SUBAPPLICATION SoftKey_Kurz_Lang (* Unterscheidet kurzen Tastendruck (Loslassen vor Ablauf PT) von langem Tastendruck (PT gehalten) auf einem AX-Adapter-Eingang (z.B. Softkey_IXA.IN). LANG feuert sofort beim Erreichen von PT (nicht erst beim Loslassen); KURZ feuert beim Loslassen, wenn PT noch nicht erreicht war. PT konfigurierbar (Parameter, Default 5s). *)
  (* Standard: 61499-2; Description: Copyright (c) 2026 Meisterschulen am Ostbahnhof This program and the accompanying materials are made available under the terms of the Eclipse Public License 2.0 which is available at https://www.eclipse.org/legal/epl-2.0/ SPDX-License-Identifier: EPL-2.0 *)
  (* Version 2.0, 2026-09-11, Franz Höpfinger, Meisterschulen am Ostbahnhof, PT konfigurierbar gemacht (Parameter statt fest 5s), umbenannt von SoftKey_Kurz_Lang_5s. Race-Bug behoben: PERMIT_KURZ pruefte bisher E_TON.Q im selben Loslass-Event, das E_TON.Q durch denselben IN-Flankenwechsel bereits auf FALSE zuruecksetzt - KURZ waere dadurch IMMER durchgelassen worden, auch nach bereits gefeuertem LANG (Ausfuehrungsreihenfolge zwischen E_TON und F_TRIG_RELEASE auf denselben IN-Event ist nicht garantiert/nicht das Kriterium). Neu: eigener LANG_LATCH (AX_SR), gesetzt durch R_TRIG_LONG (waehrend PT noch gehalten wird, zeitlich klar vor jedem Loslassen), zurueckgesetzt erst beim naechsten Tastendruck-Start (R_TRIG_PRESS) - PERMIT_KURZ prueft jetzt diesen Latch statt E_TON.Q direkt. Ausserdem SPLIT_IN (AX_SPLIT_3) ergaenzt: IN wird auf 3 Sockets (E_TON/R_TRIG_PRESS/F_TRIG_RELEASE) verteilt - ein AX-Socket darf nicht direkt auf mehrere Ziel-Sockets verbunden werden, dafuer gibt es die AX_SPLIT_n-Familie. *)
  (* Version 1.0, 2026-09-11, Franz Höpfinger, Meisterschulen am Ostbahnhof, initial implementation - fuer Achslenkung-Mittelpunkt-Taste (kurz=Anfahren, lang=Speichern), generisch fuer jede Softkey-Kurz/Lang-Unterscheidung *)
  PACKAGE MyLib::sys;
  (* Documentation:
  Kurz/Lang-Druck-Unterscheidung (konfigurierbare Haltezeit)
   E_TON (AX_TON, PT als Parameter/InputVar konfigurierbar, Default 5s) laeuft solange IN gehalten wird. R_TRIG_LONG erkennt die steigende Flanke von E_TON.Q - das ist der Moment, in dem PT erreicht ist, waehrend die Taste noch gehalten wird - und feuert LANG sofort, ohne auf das Loslassen zu warten. Gleichzeitig setzt R_TRIG_LONG den LANG_LATCH (AX_SR).
   F_TRIG_RELEASE erkennt die fallende Flanke von IN (Loslassen). PERMIT_KURZ (AX_E_PERMIT_INVERT_1) laesst dieses Ereignis nur durch, wenn LANG_LATCH.Q zu diesem Zeitpunkt FALSE ist - also wenn LANG in diesem Tastendruck-Zyklus noch nicht gefeuert wurde. LANG_LATCH wird beim naechsten Tastendruck-Start (R_TRIG_PRESS) wieder zurueckgesetzt.
   Wichtig (Bugfix ggue. Version 1.0): die Pruefung darf NICHT direkt auf E_TON.Q erfolgen - E_TON.Q wird durch denselben IN-Flankenwechsel (Loslassen), der auch F_TRIG_RELEASE ausloest, ebenfalls auf FALSE zurueckgesetzt (AX_TON: kein IN -> kein Q). Da beide Ziele (E_TON und F_TRIG_RELEASE) vom selben IN-Event gespeist werden, ist die Ausfuehrungsreihenfolge zwischen ihnen nicht garantiert - E_TON.Q waere zum Zeitpunkt der Pruefung faktisch IMMER schon FALSE, wodurch KURZ auch nach bereits gefeuertem LANG zusaetzlich gefeuert haette. Der LANG_LATCH ist von diesem Reset-Timing komplett entkoppelt (gesetzt waehrend des Haltens, zurueckgesetzt erst beim naechsten Tastendruck) und macht die Pruefung robust.
  *)
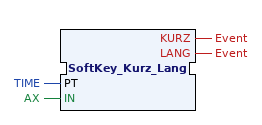
  EVENT_OUTPUT
    KURZ; (* Kurzer Druck bestaetigt (Loslassen vor Ablauf PT) *)
    LANG; (* Langer Druck bestaetigt (PT erreicht, feuert sofort - nicht erst beim Loslassen) *)
  END_EVENT
  VAR_INPUT
    PT : TIME := T#5s; (* Haltezeit fuer 'lang' *)
  END_VAR
  SOCKETS
    IN : adapter::types::unidirectional::AX; (* Rohzustand der Taste (z.B. Softkey_IXA.IN) *)
  END_SOCKETS
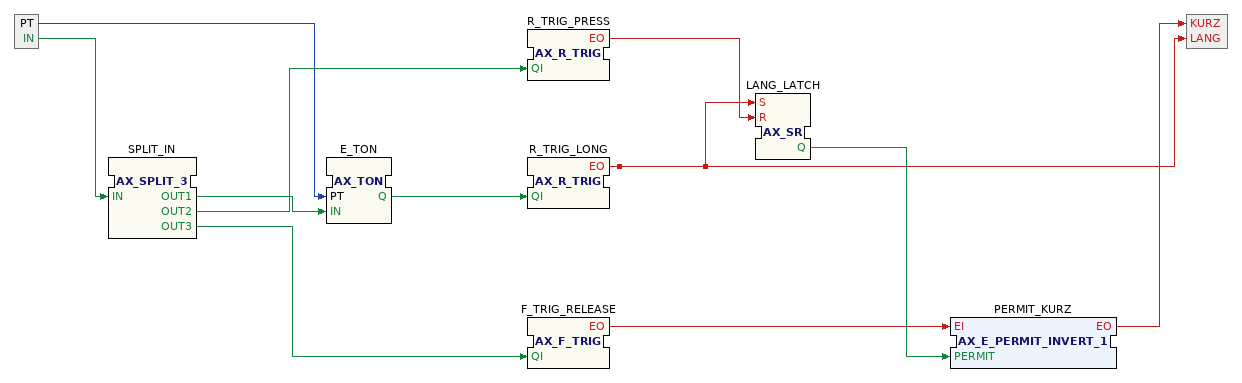
  FBS
    SPLIT_IN : adapter::events::unidirectional::AX_SPLIT_3;
    E_TON : adapter::events::unidirectional::timers::AX_TON;
    R_TRIG_LONG : adapter::events::unidirectional::AX_R_TRIG;
    R_TRIG_PRESS : adapter::events::unidirectional::AX_R_TRIG;
    LANG_LATCH : adapter::events::unidirectional::AX_SR;
    F_TRIG_RELEASE : adapter::events::unidirectional::AX_F_TRIG;
  END_FBS
  SUBAPPS
    PERMIT_KURZ : MyLib::sys::AX_E_PERMIT_INVERT_1;
  END_SUBAPPS
  EVENT_CONNECTIONS
    R_TRIG_LONG.EO TO LANG;
    R_TRIG_LONG.EO TO LANG_LATCH.S;
    R_TRIG_PRESS.EO TO LANG_LATCH.R;
    F_TRIG_RELEASE.EO TO PERMIT_KURZ.EI;
    PERMIT_KURZ.EO TO KURZ;
  END_CONNECTIONS
  DATA_CONNECTIONS
    PT TO E_TON.PT;
  END_CONNECTIONS
  ADAPTER_CONNECTIONS
    IN TO SPLIT_IN.IN;
    SPLIT_IN.OUT1 TO E_TON.IN;
    SPLIT_IN.OUT2 TO R_TRIG_PRESS.QI;
    SPLIT_IN.OUT3 TO F_TRIG_RELEASE.QI;
    E_TON.Q TO R_TRIG_LONG.QI;
    LANG_LATCH.Q TO PERMIT_KURZ.PERMIT;
  END_CONNECTIONS
END_SUBAPPLICATION
